// Mitsubishi GX Works2 project: targil2_liav   PLC: FX3G

// global labels: Global1
VAR_GLOBAL
  sw10 AT X010 : BOOL;
  inventory_good AT M10 : BOOL;
  start_stage1 AT M4 : BOOL;
  coil_10 AT Y010 : BOOL;
  sw2 AT X002 : BOOL;
  input_flour AT D1100 : REAL;
  flour_stock AT D1200 : REAL;
  input_yeast AT D1105 : REAL;
  yeast_stock AT D1205 : REAL;
  input_water AT D1110 : REAL;
  water_stock AT D1210 : REAL;
  input_oil AT D1115 : REAL;
  oil_stock AT D1215 : REAL;
  input_spices AT D1120 : REAL;
  spices_stock AT D1220 : REAL;
END_VAR
VAR_GLOBAL CONSTANT
  flour_limit : REAL := 100;
  prop1 : REAL := 0.2;
END_VAR
VAR_GLOBAL
  yeast_limit AT D1300 : REAL;
END_VAR
VAR_GLOBAL CONSTANT
  prop2 : REAL := 0.5;
END_VAR
VAR_GLOBAL
  water_limit AT D1305 : REAL;
END_VAR
VAR_GLOBAL CONSTANT
  prop3 : REAL := 0.3;
END_VAR
VAR_GLOBAL
  oil_limit AT D1310 : REAL;
END_VAR
VAR_GLOBAL CONSTANT
  prop4 : REAL := 0.1;
END_VAR
VAR_GLOBAL
  spices_limit AT D1315 : REAL;
  EMERGENCY_BUTTON AT X007 : BOOL;
  inventory_goodM AT M10 : BOOL;
  pour_time AT TC1 : BOOL;
  pour_time_TS AT TS1 : BOOL;
  coil_5 AT Y005 : BOOL;
END_VAR
VAR_GLOBAL CONSTANT
  flour_use : REAL := 100;
  yeast_use : REAL := 20;
  water_use : REAL := 50;
  oil_use : REAL := 30;
  spices_use : REAL := 10;
END_VAR
VAR_GLOBAL
  start_stage1b AT M5 : BOOL;
  sw1 AT X001 : BOOL;
  coil_1 AT Y001 : BOOL;
  double_switch AT M11 : BOOL;
  memory_double_switch AT M50 : BOOL;
  first_switch_indicator AT M50 : BOOL;
  second_switch_indicator AT M51 : BOOL;
  contact AT Y001 : BOOL;
  counter_2 AT CC0 : BOOL;
  set_2 AT M2 : BOOL;
END_VAR
VAR_GLOBAL CONSTANT
  constant_2 : INT := 2;
END_VAR
VAR_GLOBAL
  RST_C0 AT CC0 : BOOL;
  RST_Y01 AT Y001 : BOOL;
  time_2sec AT TC20 : BOOL;
END_VAR
VAR_GLOBAL CONSTANT
  time_constant : INT := 2;
END_VAR
VAR_GLOBAL
  outC AT CS0 : BOOL;
  output AT Y011 : BOOL;
  ub_limit AT S2 : BOOL;
  lb_limit AT S1 : BOOL;
  oven_works AT Y030 : BOOL;
  oven_isready AT Y003 : BOOL;
  Timer_oven AT TC3 : BOOL;
  switch1 AT M0 : BOOL;
  first_switch AT M0 : BOOL;
  TS_1 AT TS1 : BOOL;
  M_0 AT M0 : BOOL;
  tC1 AT TC1 : BOOL;
END_VAR
VAR_GLOBAL CONSTANT
  constant_05 : REAL;
  CONSTANT_1 : BOOL := 1;
END_VAR
VAR_GLOBAL
  first_lamp_oven AT M0 : BOOL;
  second_lamp_oven AT M1 : BOOL;
  Move_dough AT M150 : BOOL;
END_VAR
VAR_GLOBAL CONSTANT
  dough_container : BOOL;
END_VAR
VAR_GLOBAL
  dough AT D1400 : REAL;
  bake_time AT TC5 : BOOL;
END_VAR
VAR_GLOBAL CONSTANT
  constant_4 : INT := 4;
END_VAR
VAR_GLOBAL
  Bake_time_TS AT TS4 : BOOL;
  Bake_in_proccess AT M44 : BOOL;
  sw11 AT X011 : BOOL;
  End_day AT M20 : BOOL;
  Timer_end_day AT TC20 : BOOL;
  TS_20 AT TS20 : BOOL;
  M_21 AT M21 : BOOL;
  TS_2 AT TS2 : BOOL;
END_VAR
VAR_GLOBAL CONSTANT
  Time2 : INT := 30;
  rise_timer : INT := 30;
END_VAR
VAR_GLOBAL
  TS_4 AT TS4 : BOOL;
  coil_2 AT Y002 : BOOL;
  coil_3 AT Y003 : BOOL;
END_VAR
VAR_GLOBAL CONSTANT
  flicker_constant : INT := 2;
END_VAR
VAR_GLOBAL
  flour_stock_good AT M15 : BOOL;
  tC_2 AT TC2 : BOOL;
  tc_3 AT TC3 : BOOL;
  TS_3 AT TS3 : BOOL;
  TC_4 AT TC4 : BOOL;
  flour_good AT M15 : BOOL;
  yeast_good AT M16 : BOOL;
  water_good AT M17 : BOOL;
  oil_good AT M18 : BOOL;
  spices_good AT M19 : BOOL;
  in_stage1a AT M5 : BOOL;
END_VAR
VAR_GLOBAL CONSTANT
  bake_timer : INT := 40;
END_VAR
VAR_GLOBAL
  TC_5 AT TC5 : BOOL;
  TS_5 AT TS5 : BOOL;
  sw3 AT X003 : BOOL;
  coil_4 AT Y004 : BOOL;
  start_stage4 AT M45 : BOOL;
  finish_check AT M46 : BOOL;
  notGOOD_check AT M47 : BOOL;
END_VAR
VAR_GLOBAL CONSTANT
  MAX_quality : INT := 2000;
END_VAR
VAR_GLOBAL
  analog2 AT D8281 : INT;
  good_bread AT TC6 : BOOL;
END_VAR
VAR_GLOBAL CONSTANT
  good_bread_timer : INT := 50;
END_VAR
VAR_GLOBAL
  TS_6 AT TS6 : BOOL;
  coil_6 AT Y006 : BOOL;
  check_inventory AT M99 : BOOL;
  new_iteration AT M99 : BOOL;
  finish_bread AT M80 : BOOL;
  rising_dough AT D1410 : REAL;
  oven_container AT D1420 : REAL;
  bread_in_shelf AT D1430 : REAL;
  counter_4 AT CC1 : BOOL;
  double_check AT CS1 : BOOL;
  throw_bread AT M70 : BOOL;
  above_quality AT M91 : BOOL;
  below_quality AT M92 : BOOL;
  GOOD_check AT M47 : BOOL;
  steady_light AT M23 : BOOL;
  finish_light AT M24 : BOOL;
  end_day_time AT TC8 : BOOL;
END_VAR
VAR_GLOBAL CONSTANT
  tc8 : INT := 30;
END_VAR
VAR_GLOBAL
  TS_8 AT TS8 : BOOL;
  light_on AT TC9 : BOOL;
END_VAR
VAR_GLOBAL CONSTANT
  tc9 : INT := 2;
END_VAR
VAR_GLOBAL
  light_of AT TC10 : BOOL;
  tc10 AT TC10 : BOOL;
  BLINK AT M26 : BOOL;
  TS_9 AT TS9 : BOOL;
  TS_10 AT TS10 : BOOL;
  of_bliNk AT M27 : BOOL;
  not_above_quality AT M91 : BOOL;
  not_below_quality AT M92 : BOOL;
END_VAR

// task Task_01 (event TRUE, interval 0, priority 31): POU_01

PROGRAM POU_01
VAR CONSTANT
  pour_timer : INT := 30;
  end_timer : WORD := 2;
  MIN_quality : INT := 400;
  quantity_div : REAL := 210;
END_VAR
(* structured ladder/FBD written out as ST: instructions are called as NAME(EN, inputs, outputs); _pN, _eN, _tN stand for wires *)
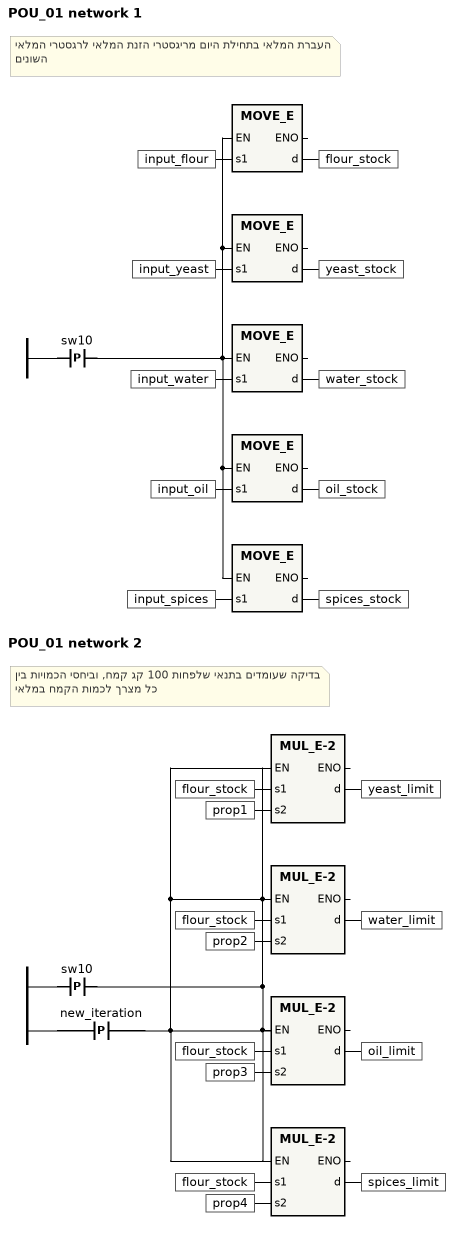
(* network 1 *)
(* העברת המלאי בתחילת היום מריגסטרי הזנת המלאי לרגסטרי המלאי השונים *)
_p1 := LDP(TRUE, sw10);
MOVE_E(_p1, input_flour, flour_stock);
MOVE_E(_p1, input_yeast, yeast_stock);
MOVE_E(_p1, input_water, water_stock);
MOVE_E(_p1, input_oil, oil_stock);
MOVE_E(_p1, input_spices, spices_stock);
(* network 2 *)
(* בדיקה שעומדים בתנאי שלפחות 100 קג קמח, וביחסי הכמויות בין כל מצרך לכמות הקמח במלאי *)
_p1 := LDP(TRUE, sw10) OR LDP(TRUE, new_iteration);
MUL_E(_p1, flour_stock, prop1, yeast_limit);
MUL_E(_p1, flour_stock, prop2, water_limit);
MUL_E(_p1, flour_stock, prop3, oil_limit);
MUL_E(_p1, flour_stock, prop4, spices_limit);
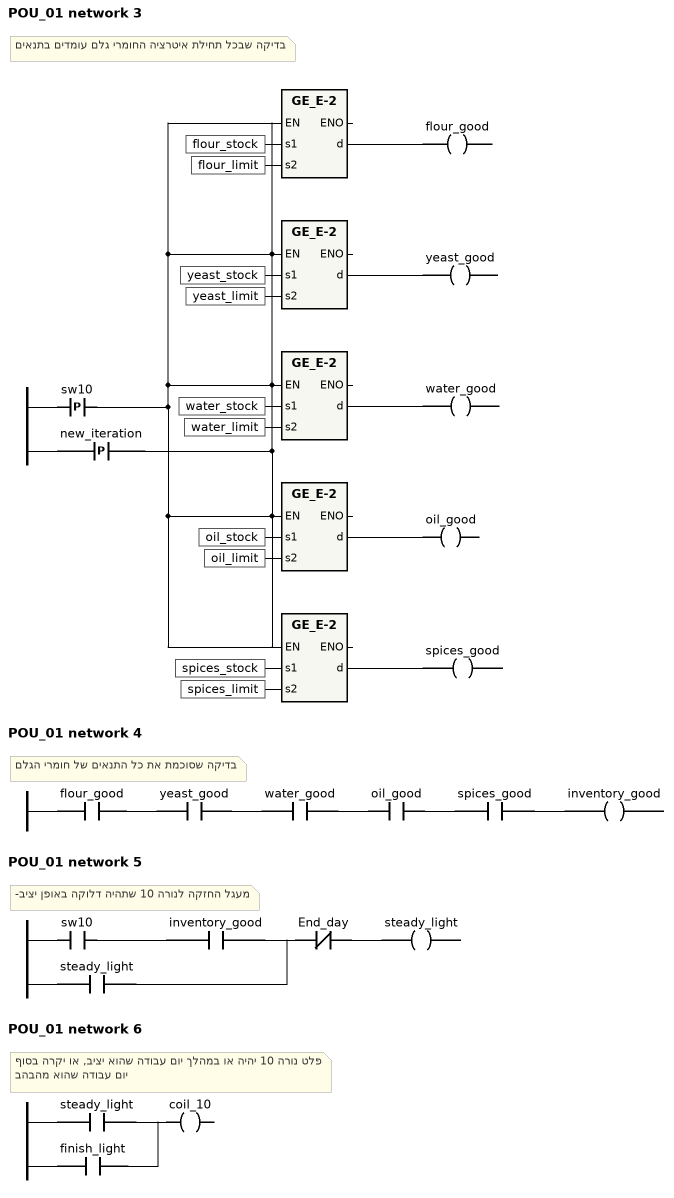
(* network 3 *)
(* בדיקה שבכל תחילת איטרציה החומרי גלם עומדים בתנאים *)
_p1 := LDP(TRUE, sw10) OR LDP(TRUE, new_iteration);
GE_E(_p1, flour_stock, flour_limit, _t2);
flour_good := _t2;
GE_E(_p1, yeast_stock, yeast_limit, _t3);
yeast_good := _t3;
GE_E(_p1, water_stock, water_limit, _t4);
water_good := _t4;
GE_E(_p1, oil_stock, oil_limit, _t5);
oil_good := _t5;
GE_E(_p1, spices_stock, spices_limit, _t6);
spices_good := _t6;
(* network 4 *)
(* בדיקה שסוכמת את כל התנאים של חומרי הגלם *)
inventory_good := flour_good AND yeast_good AND water_good AND oil_good AND spices_good;
(* network 5 *)
(* מעגל החזקה לנורה 10 שתהיה דלוקה באופן יציב- *)
steady_light := ((sw10 AND inventory_good) OR steady_light) AND NOT End_day;
(* network 6 *)
(* פלט נורה 10 יהיה או במהלך יום עבודה שהוא יציב, או יקרה בסוף יום עבודה שהוא מהבהב *)
coil_10 := steady_light OR finish_light;
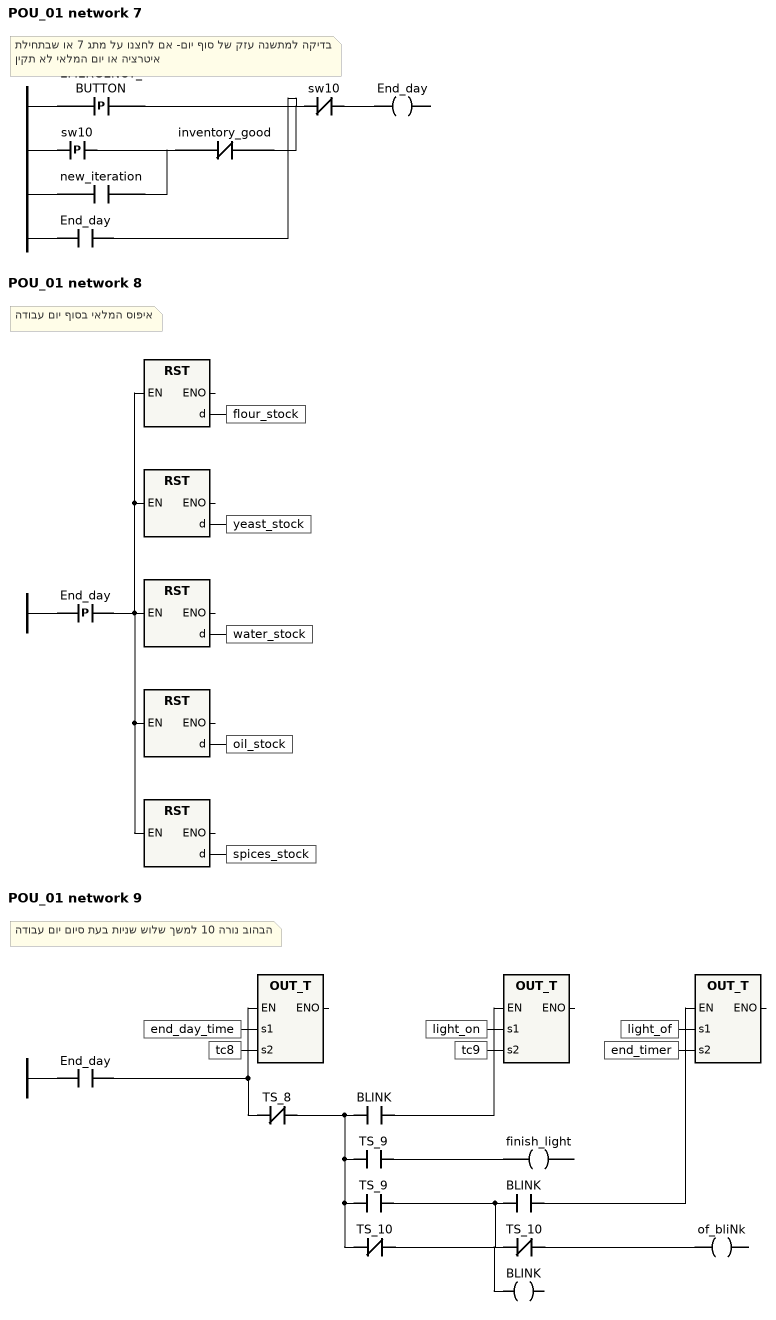
(* network 7 *)
(* בדיקה למתשנה עזק של סוף יום- אם לחצנו על מתג 7 או שבתחילת איטרציה או יום המלאי לא תקין *)
End_day := (LDP(TRUE, EMERGENCY_BUTTON) OR ((LDP(TRUE, sw10) OR new_iteration) AND NOT inventory_good) OR End_day) AND NOT sw10;
(* network 8 *)
(* איפוס המלאי בסוף יום עבודה *)
_p1 := LDP(TRUE, End_day);
RST(_p1, flour_stock);
RST(_p1, yeast_stock);
RST(_p1, water_stock);
RST(_p1, oil_stock);
RST(_p1, spices_stock);
(* network 9 *)
(* הבהוב נורה 10 למשך שלוש שניות בעת סיום יום עבודה *)
OUT_T(End_day, end_day_time, tc8);
_p1 := End_day AND NOT TS_8;
OUT_T(_p1 AND BLINK, light_on, tc9);
finish_light := _p1 AND TS_9;
_p2 := _p1 AND TS_9;
OUT_T(_p2 AND BLINK, light_of, end_timer);
of_bliNk := _p2 AND NOT TS_10;
BLINK := _p1 AND NOT TS_10;
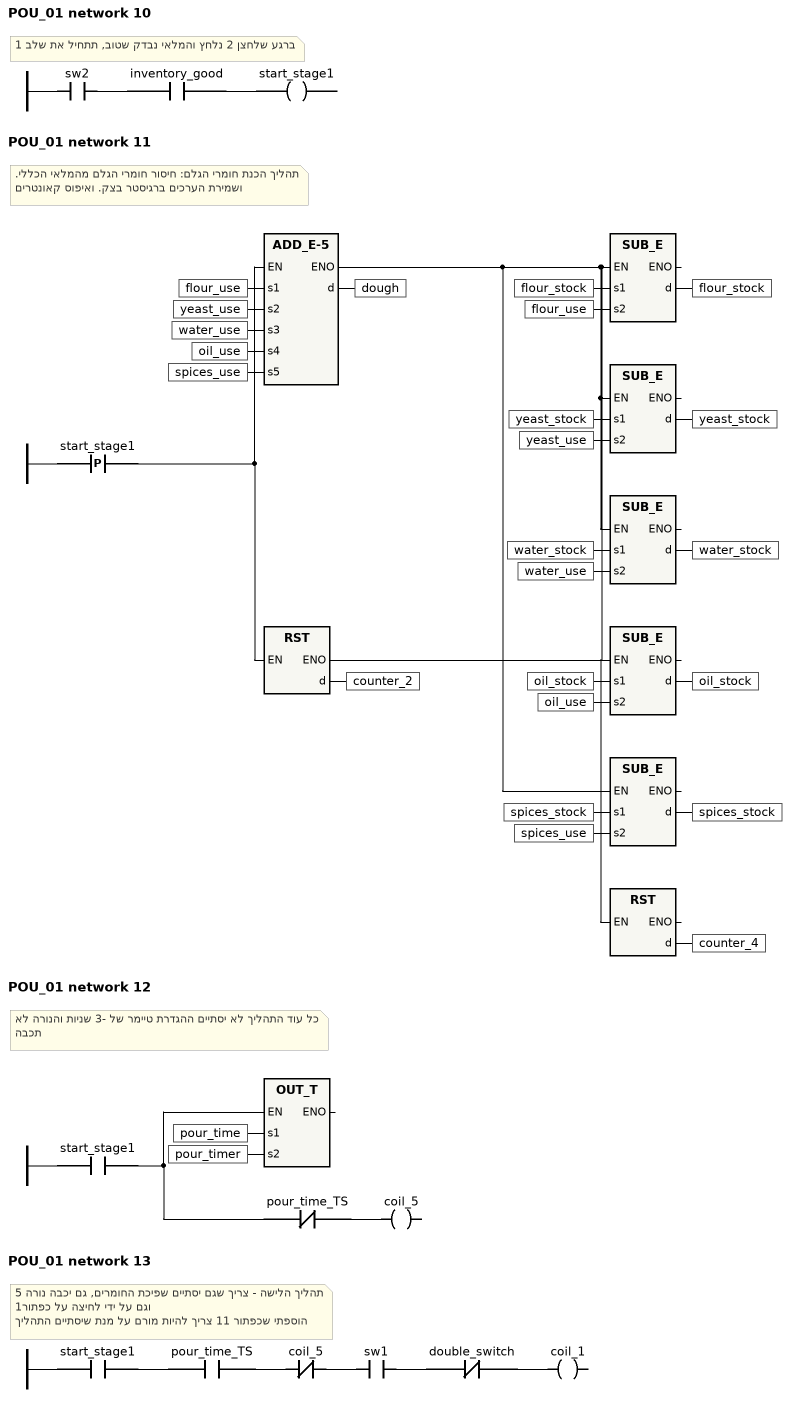
(* network 10 *)
(* ברגע שלחצן 2 נלחץ והמלאי נבדק שטוב, תתחיל את שלב 1 *)
start_stage1 := sw2 AND inventory_good;
(* network 11 *)
(* תהליך הכנת חומרי הגלם: חיסור חומרי הגלם מהמלאי הכללי. ושמירת הערכים ברגיסטר בצק. ואיפוס קאונטרים *)
_p1 := LDP(TRUE, start_stage1);
_e2 := ADD_E(_p1, flour_use, yeast_use, water_use, oil_use, spices_use, dough);
SUB_E(_e2, flour_stock, flour_use, flour_stock);
SUB_E(_e2, yeast_stock, yeast_use, yeast_stock);
SUB_E(_e2, water_stock, water_use, water_stock);
SUB_E(_e2, oil_stock, oil_use, oil_stock);
SUB_E(_e2, spices_stock, spices_use, spices_stock);
_e3 := RST(_p1, counter_2);
RST(_e3, counter_4);
(* network 12 *)
(* כל עוד התהליך לא יסתיים ההגדרת טיימר של -3 שניות והנורה לא תכבה *)
OUT_T(start_stage1, pour_time, pour_timer);
coil_5 := start_stage1 AND NOT pour_time_TS;
(* network 13 *)
(* תהליך הלישה - צריך שגם יסתיים שפיכת החומרים, גם יכבה נורה 5 וגם על ידי לחיצה על כפתור1 / הוספתי שכפתור 11 צריך להיות מורם על מנת שיסתיים התהליך *)
coil_1 := start_stage1 AND pour_time_TS AND NOT coil_5 AND sw1 AND NOT double_switch;
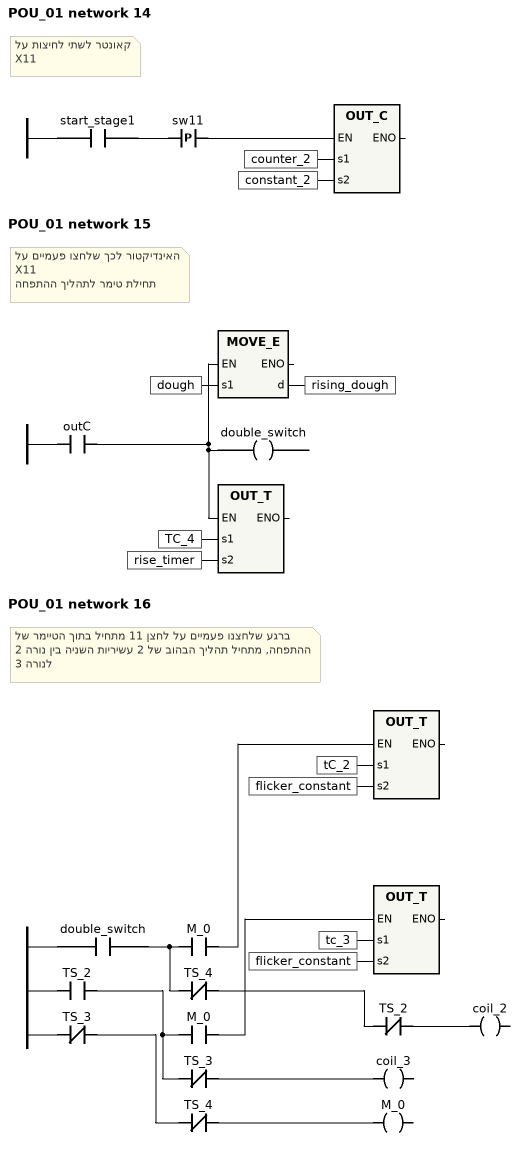
(* network 14 *)
(* קאונטר לשתי לחיצות על  / X11 *)
OUT_C(start_stage1 AND LDP(TRUE, sw11), counter_2, constant_2);
(* network 15 *)
(* האינדיקטור לכך שלחצו פעמיים על  / X11 / תחילת טימר לתהליך ההתפחה *)
MOVE_E(outC, dough, rising_dough);
double_switch := outC;
OUT_T(outC, TC_4, rise_timer);
(* network 16 *)
(* ברגע שלחצנו פעמיים על לחצן 11 מתחיל בתוך הטיימר של ההתפחה, מתחיל תהליך הבהוב של 2 עשיריות השניה בין נורה 2 לנורה 3 *)
OUT_T(double_switch AND M_0, tC_2, flicker_constant);
coil_2 := double_switch AND NOT TS_4 AND NOT TS_2;
OUT_T(TS_2 AND M_0, tc_3, flicker_constant);
coil_3 := TS_2 AND NOT TS_3;
M_0 := NOT TS_3 AND NOT TS_4;
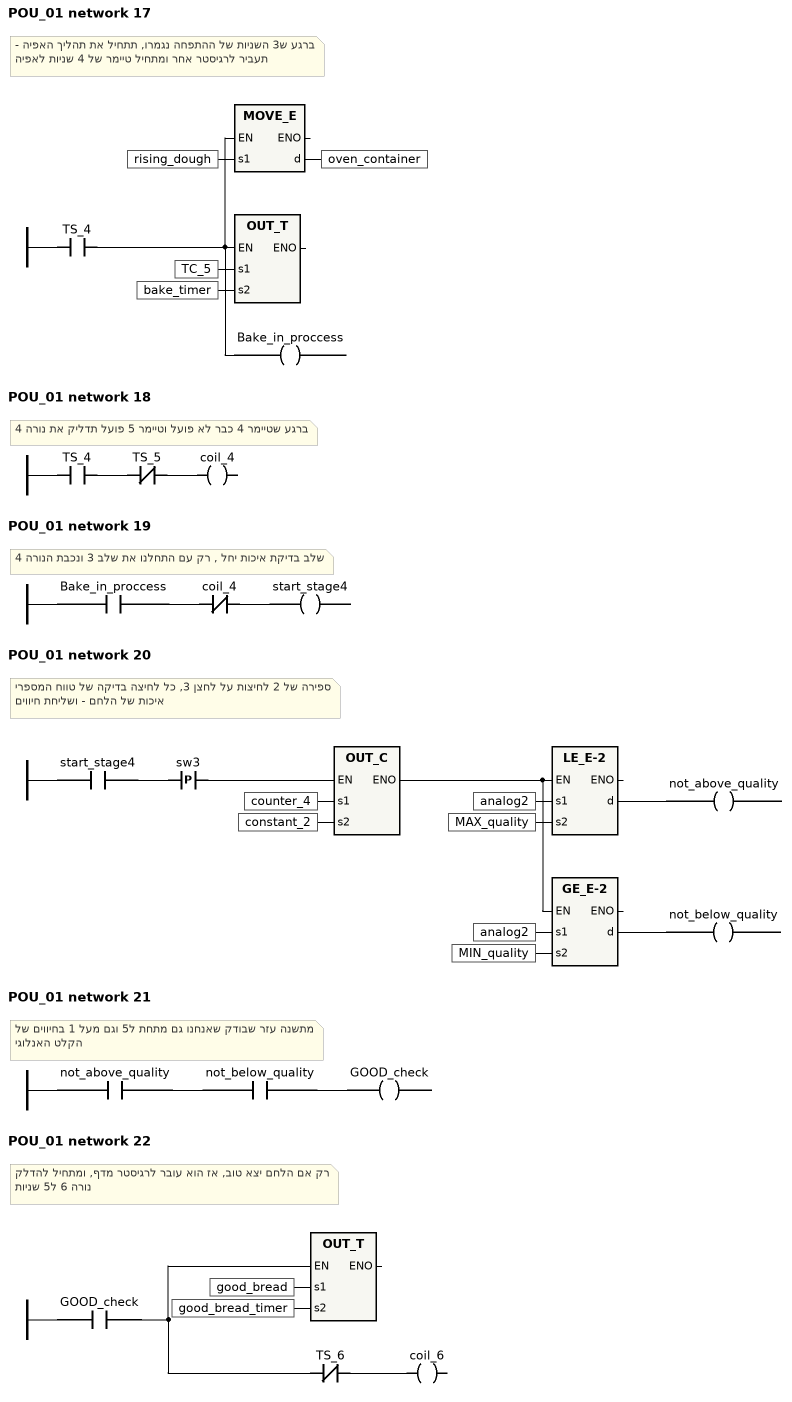
(* network 17 *)
(* ברגע ש3 השניות של ההתפחה נגמרו, תתחיל את תהליך האפיה - תעביר לרגיסטר אחר ומתחיל טיימר של 4 שניות לאפיה *)
MOVE_E(TS_4, rising_dough, oven_container);
OUT_T(TS_4, TC_5, bake_timer);
Bake_in_proccess := TS_4;
(* network 18 *)
(* ברגע שטיימר 4 כבר לא פועל וטיימר 5 פועל תדליק את נורה 4 *)
coil_4 := TS_4 AND NOT TS_5;
(* network 19 *)
(* שלב בדיקת איכות יחל , רק עם התחלנו את שלב 3 ונכבת הנורה 4 *)
start_stage4 := Bake_in_proccess AND NOT coil_4;
(* network 20 *)
(* ספירה של 2 לחיצות על לחצן 3, כל לחיצה בדיקה של טווח המספרי איכות של הלחם - ושליחת חיווים *)
_e1 := OUT_C(start_stage4 AND LDP(TRUE, sw3), counter_4, constant_2);
LE_E(_e1, analog2, MAX_quality, _t2);
not_above_quality := _t2;
GE_E(_e1, analog2, MIN_quality, _t3);
not_below_quality := _t3;
(* network 21 *)
(* מתשנה עזר שבודק שאנחנו גם מתחת ל5 וגם מעל 1 בחיווים של הקלט האנלוגי *)
GOOD_check := not_above_quality AND not_below_quality;
(* network 22 *)
(* רק אם הלחם יצא טוב, אז הוא עובר לרגיסטר מדף, ומתחיל להדלק נורה 6 ל5 שניות *)
OUT_T(GOOD_check, good_bread, good_bread_timer);
coil_6 := GOOD_check AND NOT TS_6;
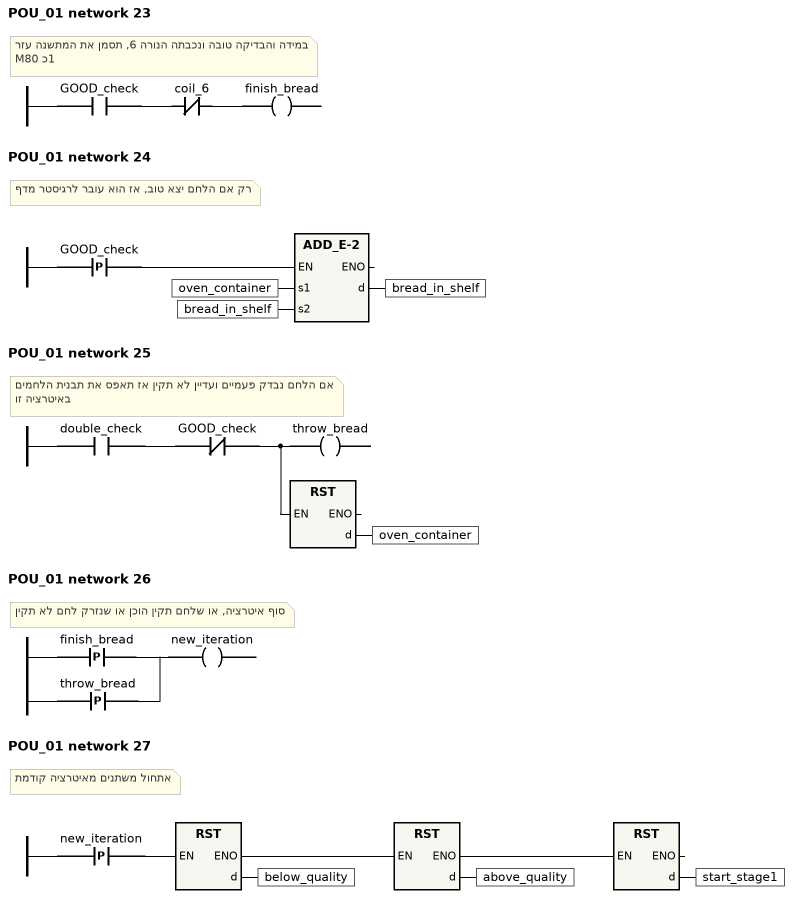
(* network 23 *)
(* במידה והבדיקה טובה ונכבתה הנורה 6, תסמן את המתשנה עזר M80 כ1 *)
finish_bread := GOOD_check AND NOT coil_6;
(* network 24 *)
(* רק אם הלחם יצא טוב, אז הוא עובר לרגיסטר מדף *)
ADD_E(LDP(TRUE, GOOD_check), oven_container, bread_in_shelf, bread_in_shelf);
(* network 25 *)
(* אם הלחם נבדק פעמיים ועדיין לא תקין אז תאפס את תבנית הלחמים באיטרציה זו *)
_p1 := double_check AND NOT GOOD_check;
throw_bread := _p1;
RST(_p1, oven_container);
(* network 26 *)
(* סוף איטרציה, או שלחם תקין הוכן או שנזרק לחם לא תקין *)
new_iteration := LDP(TRUE, finish_bread) OR LDP(TRUE, throw_bread);
(* network 27 *)
(* אתחול משתנים מאיטרציה קודמת *)
_e1 := RST(LDP(TRUE, new_iteration), below_quality);
_e2 := RST(_e1, above_quality);
RST(_e2, start_stage1);
END_PROGRAM
